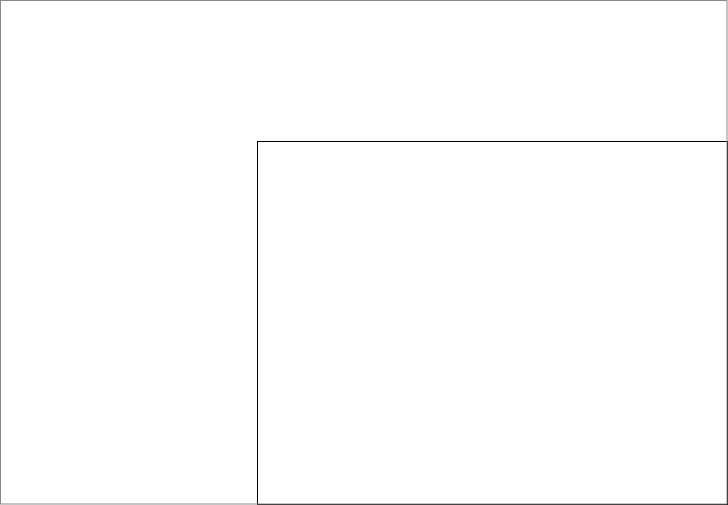
VISUALIZATION Visualization  // 728x505
    Rectangle (257,141 471x364)
END_VISUALIZATION

(* stored: Version 1.1.0.1, ProductVersion 3.1.4024.12
   Visu Visualization: Id {8096fc08-ffd6-4f12-b0e7-66246e50a2f3} *)
